// TIA Portal V20 export
FUNCTION "Limit Mapping" : Void   // FC105, SCL
{ S7_Optimized_Access := 'TRUE' }
// stored: SetENOAutomatically false
   VAR_INPUT
      Limit_Sensor1 : Bool;
      Limit_Sensor2 : Bool;
      Limit_Sensor3 : Bool;
      Limit_Sensor4 : Bool;
      Limit_Sensor5 : Bool;
      Limit_Sensor6 : Bool;
      Limit_Sensor7 : Bool;
      Limit_Sensor8 : Bool;
   END_VAR
   VAR_OUTPUT
      O_Sensor1 : Bool;
      O_Sensor2 : Bool;
      O_Sensor3 : Bool;
      O_Sensor4 : Bool;
      O_Sensor5 : Bool;
      O_Sensor6 : Bool;
      O_Sensor7 : Bool;
      O_Sensor8 : Bool;
   END_VAR
BEGIN
   #O_Sensor1 := #Limit_Sensor1;
   #O_Sensor2 := #Limit_Sensor2;
   #O_Sensor3 := #Limit_Sensor3;
   #O_Sensor4 := #Limit_Sensor4;
   #O_Sensor5 := #Limit_Sensor5;
   #O_Sensor6 := #Limit_Sensor6;
   #O_Sensor7 := #Limit_Sensor7;
   #O_Sensor8 := #Limit_Sensor8;
END_FUNCTION
